FUNCTION_BLOCK UA_NodeGetHandleWrapper IMPLEMENTS I_OPCUA_NodeGetHandle
VAR_INPUT
END_VAR
VAR_OUTPUT
END_VAR
VAR
	uaNodegethandle : UA_NodeGetHandle;
END_VAR

{warning 'add method implementation '}
METHOD start : BOOL
VAR_INPUT
	Execute	: BOOL;
	ConnectionHdl	: DWORD;
	NodeID	: Tc3_PLCopen_OpcUa.ST_UANodeID;
	Timeout	: TIME := DEFAULT_ADS_TIMEOUT;
END_VAR
VAR_OUTPUT
	NodeHdl	: DWORD;
	Done	: BOOL;
	Busy	: BOOL;
	Error	: BOOL;
	ErrorID	: DWORD;
END_VAR
uaNodegethandle(Execute := execute, 
				connectionhdl := connectionhdl, 
				nodeid := nodeid, 
				timeout := timeout,
				NodeHdl => NodeHdl,
				Done => Done,
				Busy => Busy,
				Error => Error,
				ErrorID => ErrorId);
END_METHOD

END_FUNCTION_BLOCK

(* stored: Version 1.1.0.1, ProductVersion 3.1.4024.9
   POU UA_NodeGetHandleWrapper: Id {d32f359d-c4d0-4e45-8062-bdf901152801}, SpecialFunc None
   Method start: Id {c67e8e69-01af-43c8-b6df-46caeb4334bc} *)
